KUKA KRL data list: SONG_2.dat

&ACCESS RVO1
DEFDAT SONG_2
;FOLD EXTERNAL DECLARATIONS;%{PE}%MKUKATPBASIS,%CEXT,%VCOMMON,%P
;FOLD BASISTECH EXT;%{PE}%MKUKATPBASIS,%CEXT,%VEXT,%P
EXT  BAS (BAS_COMMAND  :IN,REAL  :IN )
DECL INT BAR
DECL INT COUNTER
;ENDFOLD (BASISTECH EXT)
;FOLD USER EXT;%{E}%MKUKATPUSER,%CEXT,%VEXT,%P
;Make your modifications here

;ENDFOLD (USER EXT)
;ENDFOLD (EXTERNAL DECLARATIONS)
DECL MODULEPARAM_T LAST_TP_PARAMS = {PARAMS[] "Kuka.Logics.Io=1; Kuka.Logics.IoName=; Kuka.Logics.State=True; Kuka.Logics.Cont=False; Kuka.Logics.Time=0.1"}
ENDDAT
